Staubli VAL3: setAllBlend.pgx

public program setAllBlend(num x_nNewValue, num x_nOldValue)
  local num i
  local num l_nSize
begin
end
